ABB RAPID module: Part_6.mod

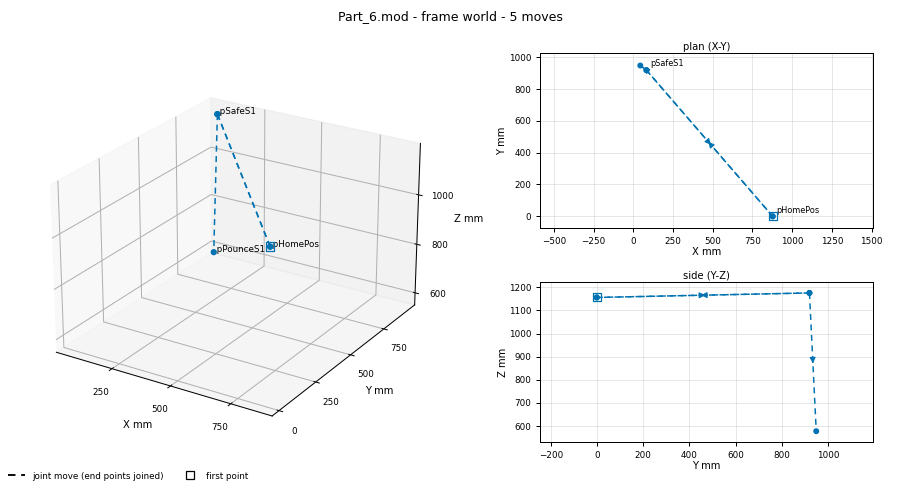
[picture p0: tool path of Part_6.mod in frame world, 5 of 13 moves have a stored position in this frame; points joined in program order, loops and branches not executed]
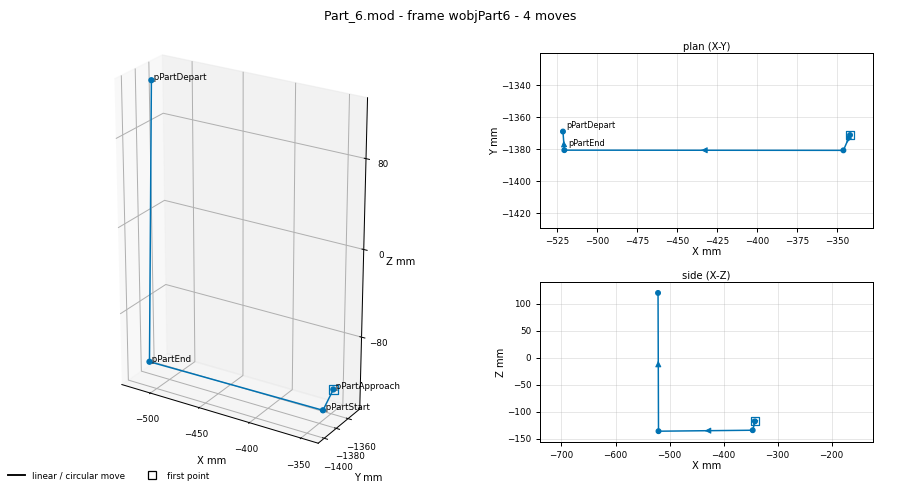
[picture p1: tool path of Part_6.mod in frame wobjPart6, 4 of 13 moves have a stored position in this frame; points joined in program order, loops and branches not executed]
MODULE Part_6
  ! ------------------------------------------------------------------
  ! Single-part welding template
  !
  ! Purpose:
  !   - Run one part only (no multi-part branching)
  !   - Keep nozzle cleaning and BullsEye tool check available
  !   - Provide a copy/paste starting point for new part files
  !
  ! Dependencies:
  !   - LogicZ (home/safe/pounce positions + rTC2013)
  !   - BE_User1 (BECheckToolb for BullsEye)
  !   - mTSC (optional torch cleaner if you prefer MechCleanGun)
  ! ------------------------------------------------------------------

  LOCAL PERS bool bUseTorchClean := TRUE;
  LOCAL PERS bool bUseBullseye := TRUE;

  ! Placeholder weld/seam data for the template. Replace with real values.
  LOCAL PERS welddata weldPart := [0,0,[1,0,0,0,0,0,0,0,0],[0,0,0,0,0,0,0,0,0]];
  LOCAL PERS seamdata seamPart := [1,1,[1,0,0,0,0,0,0,0,0],0,0,0,0,0,[0,0,0,0,0,0,0,0,0],0,0,[0,0,0,0,0,0,0,0,0],0,0,[0,0,0,0,0,0,0,0,0],0];

  ! Placeholder targets for the weld path. Replace with taught points.
  LOCAL CONST robtarget pPartApproach := [[-341.99,-1371.18,-117.57],[0.232266,0.668561,-0.669899,0.224308],[-2,-1,1,0],[9E+09,9E+09,9E+09,9E+09,9E+09,9E+09]];
  CONST robtarget pPartStart := [[-346.14,-1380.75,-134.00],[0.232258,0.668629,-0.669841,0.22429],[-2,-1,1,0],[9E+09,9E+09,9E+09,9E+09,9E+09,9E+09]];
  CONST robtarget pPartEnd := [[-520.49,-1380.63,-135.80],[0.232194,0.668749,-0.669754,0.224259],[-2,-1,1,0],[9E+09,9E+09,9E+09,9E+09,9E+09,9E+09]];
  CONST robtarget pPartDepart := [[-521.34,-1368.99,120.05],[0.232497,0.668664,-0.669682,0.22441],[-2,-1,1,0],[9E+09,9E+09,9E+09,9E+09,9E+09,9E+09]];
  PROC RunPart_6()
    TPWrite "Single-part template start";

    ! Optional BullsEye tool check before running a part.
    IF bUseBullseye THEN
      BECheckToolb;
    ENDIF

    ! Optional nozzle cleaning/reaming before the part weld.
    IF bUseTorchClean THEN
      rTC2013;
      ! Alternative: MechCleanGun;  ! From mTSC.mod
    ENDIF

    MoveJ pHomePos, v800, fine, tWeldGun;
    MoveJ pSafeS1, v800, fine, tWeldGun;
    MoveJ pPounceS1, v800, fine, tWeldGun;

    ! ----------------------------------------------------------------
    ! Single-part weld path (edit only the weld start/end points).
    ! ----------------------------------------------------------------
    IF bDryRun THEN
      MoveL DryRunTarget(pPartApproach), v200, z10, tWeldGun\WObj:=wobjPart6;
      MoveL DryRunTarget(pPartStart), v200, z10, tWeldGun\WObj:=wobjPart6;
      MoveL DryRunTarget(pPartEnd), v200, z10, tWeldGun\WObj:=wobjPart6;
      MoveL DryRunTarget(pPartDepart), v200, z10, tWeldGun\WObj:=wobjPart6;
    ELSE
      MoveL pPartApproach, v200, z10, tWeldGun\WObj:=wobjPart6;
      ArcLStart pPartStart, v30, seamPart, weldPart, fine, tWeldGun\WObj:=wobjPart6;
      ArcLEnd pPartEnd, v30, seamPart, weldPart, fine, tWeldGun\WObj:=wobjPart6;
      MoveL pPartDepart, v200, z10, tWeldGun\WObj:=wobjPart6;
    ENDIF

    MoveJ pSafeS1, v800, fine, tWeldGun;
    MoveJ pHomePos, v800, fine, tWeldGun;

    TPWrite "Single-part template complete";
  ENDPROC
ENDMODULE
